// TIA Portal V20 export
TYPE "Position"
   STRUCT
      LinAxis : Struct   // Assi lineari
         X : Real;
         Y : Real;
         Z : Real;
      END_STRUCT;
      AngAxis : Struct   // Assi angolari
         "B" : Real;
         C : Real;
      END_STRUCT;
   END_STRUCT;
END_TYPE
